// TIA Portal project "lab4" (V17)

(* hardware
DEVICE "S7-1200 station_1"  S7-1200 Station
   slot 0: "Rack_0"  S7-1200 Rack  Rack  V1.0
   slot 1: "PLC_1"  CPU 1214C DC/DC/DC  6ES7 214-1AG40-0XB0  V4.5
*)

// ===== PLC "PLC_1"  CPU 1214C DC/DC/DC =====

VAR_GLOBAL   // PLC tag table "Default tag table"
   "Zmienna_Int" AT %MW50 : Int;
   "Zmienna_Real" AT %MD52 : Real;
   "Zmienna_Word" AT %MW56 : Word;
   "Zmienna_UInt" AT %MW58 : UInt;
   "Zmienna_DInt" AT %MD59 : DInt;
   "Tag_1" AT %Q0.0 : Bool;
   "Tag_2" AT %M50.0 : Bool;
   "Tag_3" AT %M100.0 : Bool;
   "Tag_4" AT %M99.0 : Bool;
   "Tag_5" AT %Q0.1 : Bool;
   "Tag_6" AT %I0.0 : Bool;
   "Tag_7" AT %M0.0 : Bool;
   "Tag_8" AT %M0.1 : Bool;
   "Tag_9" AT %Q0.2 : Bool;
   "Tag_10" AT %IB0 : Byte;
   "Tag_11" AT %QB0 : Byte;
END_VAR

DATA_BLOCK "Rejestr_przesuwny_DB"   // DB6
{ S7_Optimized_Access := 'TRUE' }
VERSION : 0.1
   VAR
      Rejestr : Array[0..9] of Byte;
   END_VAR
BEGIN
END_DATA_BLOCK

// folder: System blocks/Program resources

DATA_BLOCK "IEC_Timer_0_DB"   // DB1
{ S7_Optimized_Access := 'TRUE' }
AUTHOR : Simatic
FAMILY : IEC
NAME : IEC_TMR
VERSION : 1.0
// stored: InstanceOfName IEC_TIMER
"IEC_TIMER"
BEGIN
END_DATA_BLOCK

DATA_BLOCK "IEC_Timer_0_DB_1"   // DB2
{ S7_Optimized_Access := 'TRUE' }
AUTHOR : Simatic
FAMILY : IEC
NAME : IEC_TMR
VERSION : 1.0
// stored: InstanceOfName IEC_TIMER
"IEC_TIMER"
BEGIN
END_DATA_BLOCK

DATA_BLOCK "IEC_Counter_0_DB"   // DB3
{ S7_Optimized_Access := 'TRUE' }
AUTHOR : Simatic
FAMILY : IEC
NAME : CNTR
VERSION : 1.0
// stored: InstanceOfName IEC_COUNTER
"IEC_COUNTER"
BEGIN
END_DATA_BLOCK

DATA_BLOCK "Counter_czerwone_DB"   // DB4
{ S7_Optimized_Access := 'TRUE' }
AUTHOR : Simatic
FAMILY : IEC
NAME : CNTR
VERSION : 1.0
// stored: InstanceOfName IEC_COUNTER
"IEC_COUNTER"
BEGIN
END_DATA_BLOCK

DATA_BLOCK "Counter_nieb_DB"   // DB5
{ S7_Optimized_Access := 'TRUE' }
AUTHOR : Simatic
FAMILY : IEC
NAME : CNTR
VERSION : 1.0
// stored: InstanceOfName IEC_COUNTER
"IEC_COUNTER"
BEGIN
END_DATA_BLOCK

// folder: (top level)

FUNCTION "2Hz" : Void   // FC1, LAD
{ S7_Optimized_Access := 'TRUE' }
VERSION : 0.1
   VAR_INPUT
      Okres : DInt;
      "Wypelnienie [%]" : Int;
   END_VAR
   VAR_OUTPUT
      OUT : Bool;
   END_VAR
   VAR_TEMP
      Wypelnienie_temp : DInt;
      Wypelnienie_DInt : DInt;
      TP_temp : Bool;
   END_VAR
   VAR_TEMP   // added for the SCL form of the ladder/FBD networks
      _w1 : Bool;
   END_VAR
BEGIN

REGION Network 1
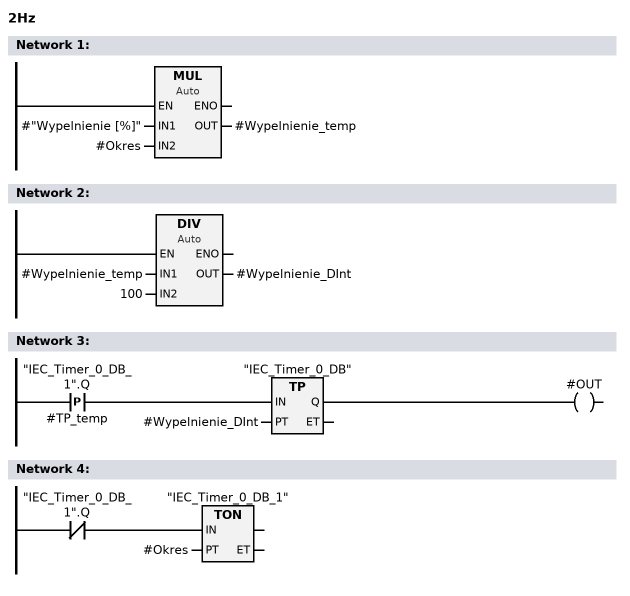
   RUNG wire#powerrail
      Mul(in1 := #"Wypelnienie [%]", in2 := #Okres, out => #Wypelnienie_temp)
   END_RUNG
   // the same network as SCL:
   #Wypelnienie_temp := #"Wypelnienie [%]" * #Okres;
END_REGION

REGION Network 2
   RUNG wire#powerrail
      Div(in1 := #Wypelnienie_temp, in2 := 100, out => #Wypelnienie_DInt)
   END_RUNG
   // the same network as SCL:
   #Wypelnienie_DInt := #Wypelnienie_temp / 100;
END_REGION

REGION Network 3
   #_w1 := "IEC_Timer_0_DB_1".Q AND NOT #TP_temp;   // rising edge of "IEC_Timer_0_DB_1".Q
   #TP_temp := "IEC_Timer_0_DB_1".Q;
   "IEC_Timer_0_DB".TP(IN := #_w1, PT := #Wypelnienie_DInt);
   #OUT := "IEC_Timer_0_DB".Q;
END_REGION

REGION Network 4
   "IEC_Timer_0_DB_1".TON(IN := NOT "IEC_Timer_0_DB_1".Q, PT := #Okres);
END_REGION
END_FUNCTION

FUNCTION "Pakowanie" : Void   // FC2, LAD
{ S7_Optimized_Access := 'TRUE' }
VERSION : 0.1
   VAR_INPUT
      Czujnik_podajnik : Bool;
      Clock : Bool;
   END_VAR
   VAR_IN_OUT
      Naped : Bool;
      Czerwony_element : Bool;
      Niebieski_element : Bool;
      Fotokomorka_nieb : Bool;
      Fotokomorka_czerw : Bool;
   END_VAR
   VAR_TEMP
      Uruchom_temp : Bool;
      Clock_temp : Bool;
      Dodaj_czerw : Bool;
      Dodaj_nieb : Bool;
   END_VAR
   VAR_TEMP   // added for the SCL form of the ladder/FBD networks
      _w1 : Bool;
   END_VAR
BEGIN

REGION Network 1
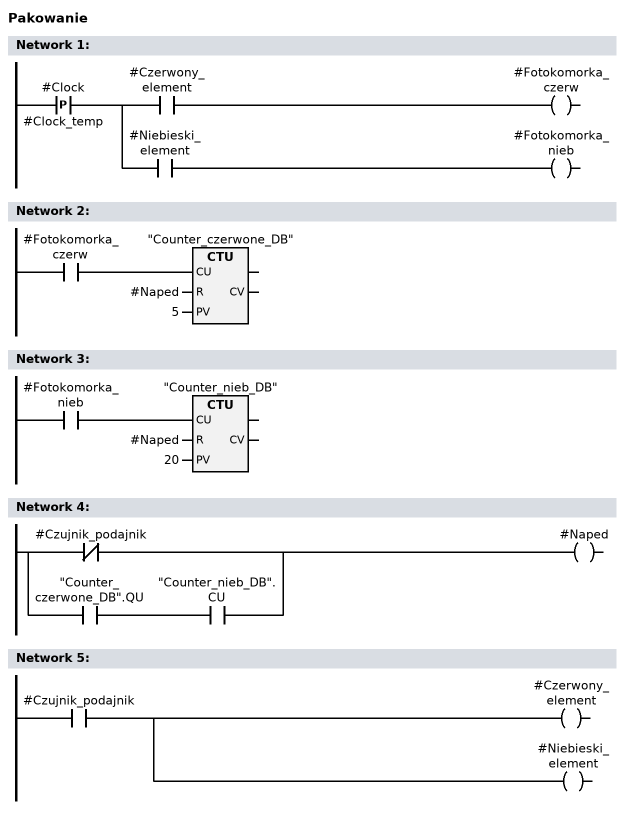
   RUNG wire#powerrail
      P_Contact(operand := #Clock, bit := #Clock_temp)
      wire#w1
      Contact( #Czerwony_element )
      Coil( #Fotokomorka_czerw )
   END_RUNG
   RUNG wire#w1
      Contact( #Niebieski_element )
      Coil( #Fotokomorka_nieb )
   END_RUNG
   // the same network as SCL:
   #_w1 := #Clock AND NOT #Clock_temp;   // rising edge of #Clock
   #Clock_temp := #Clock;
   #Fotokomorka_czerw := #_w1 AND #Czerwony_element;
   #Fotokomorka_nieb := #_w1 AND #Niebieski_element;
END_REGION

REGION Network 2
   "Counter_czerwone_DB".CTU(CU := #Fotokomorka_czerw, R := #Naped, PV := 5);
END_REGION

REGION Network 3
   "Counter_nieb_DB".CTU(CU := #Fotokomorka_nieb, R := #Naped, PV := 20);
END_REGION

REGION Network 4
   RUNG wire#powerrail
      I_Contact( #Czujnik_podajnik )
      wire#w1
      Coil( #Naped )
   END_RUNG
   RUNG wire#powerrail
      Contact( "Counter_czerwone_DB".QU )
      Contact( "Counter_nieb_DB".CU )
   END_RUNG wire#w1
   // the same network as SCL:
   #Naped := NOT #Czujnik_podajnik OR ("Counter_czerwone_DB".QU AND "Counter_nieb_DB".CU);
END_REGION

REGION Network 5
   RUNG wire#powerrail
      Contact( #Czujnik_podajnik )
      wire#w1
      Coil( #Czerwony_element )
   END_RUNG
   RUNG wire#w1
      Coil( #Niebieski_element )
   END_RUNG
   // the same network as SCL:
   #Czerwony_element := #Czujnik_podajnik;
   #Niebieski_element := #Czujnik_podajnik;
END_REGION
END_FUNCTION

FUNCTION "Dzielnik_4_1" : Void   // FC3, LAD
{ S7_Optimized_Access := 'TRUE' }
VERSION : 0.1
   VAR_INPUT
      Signal_IN : Bool;
   END_VAR
   VAR_OUTPUT
      Signal_Out : Bool;
   END_VAR
BEGIN

REGION Network 1
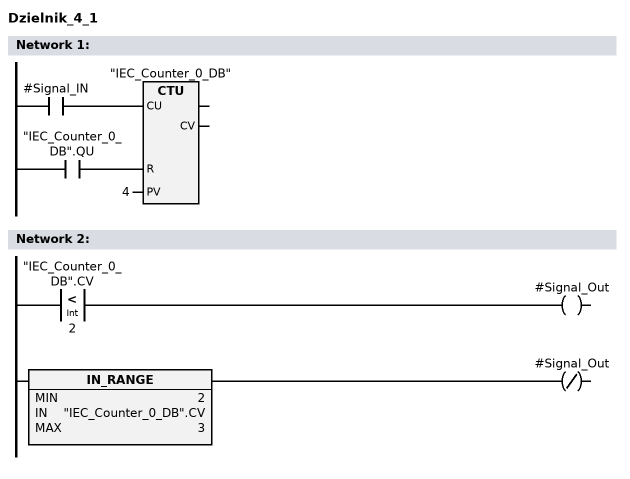
   "IEC_Counter_0_DB".CTU(CU := #Signal_IN, R := "IEC_Counter_0_DB".QU, PV := 4);
END_REGION

REGION Network 2
   RUNG wire#powerrail
      { S7_Templates := "SrcType := Int" } LT_Contact(in1 := "IEC_Counter_0_DB".CV, in2 := 2)
      Coil( #Signal_Out )
   END_RUNG
   RUNG wire#powerrail
      { S7_Templates := "SrcType := Int" } InRange(min := 2, in := "IEC_Counter_0_DB".CV, max := 3)
      I_Coil( #Signal_Out )
   END_RUNG
   // the same network as SCL:
   #Signal_Out := "IEC_Counter_0_DB".CV < 2;
   #Signal_Out := NOT ((2 <= "IEC_Counter_0_DB".CV) AND ("IEC_Counter_0_DB".CV <= 3));
END_REGION
END_FUNCTION

FUNCTION "Rejestr_przesuwny" : Void   // FC4, LAD
{ S7_Optimized_Access := 'TRUE' }
VERSION : 0.1
   VAR_INPUT
      Clock : Bool;
   END_VAR
   VAR_TEMP
      Clock_temp : Bool;
   END_VAR
   VAR_TEMP   // added for the SCL form of the ladder/FBD networks
      _w1 : Bool;
   END_VAR
BEGIN

REGION Network 1
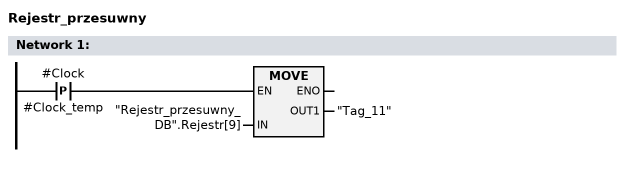
   RUNG wire#powerrail
      P_Contact(operand := #Clock, bit := #Clock_temp)
      Move(in := "Rejestr_przesuwny_DB".Rejestr[9], out1 => "Tag_11")
   END_RUNG
   // the same network as SCL:
   #_w1 := #Clock AND NOT #Clock_temp;   // rising edge of #Clock
   #Clock_temp := #Clock;
   IF #_w1 THEN "Tag_11" := "Rejestr_przesuwny_DB".Rejestr[9]; END_IF;
END_REGION
END_FUNCTION

ORGANIZATION_BLOCK "Main"   // OB1, LAD, ProgramCycle
TITLE = "Main Program Sweep (Cycle)"
{ S7_Optimized_Access := 'TRUE' }
VERSION : 0.1
   VAR_INPUT
      Initial_Call : Bool;   // Initial call of this OB
      Remanence : Bool;   // =True, if remanent data are available
   END_VAR
BEGIN

REGION Network 1
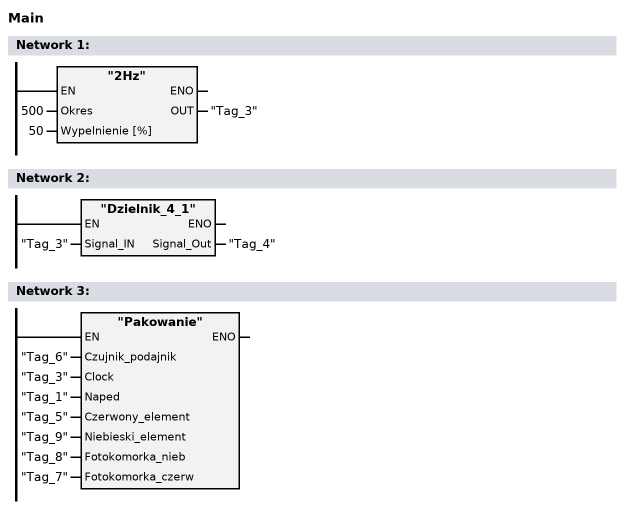
   RUNG wire#powerrail
      "2Hz"(Okres := 500, "Wypelnienie [%]" := 50, OUT => "Tag_3")
   END_RUNG
   // the same network as SCL:
   "2Hz"(Okres := 500, "Wypelnienie [%]" := 50, OUT => "Tag_3");
END_REGION

REGION Network 2
   RUNG wire#powerrail
      "Dzielnik_4_1"(Signal_IN := "Tag_3", Signal_Out => "Tag_4")
   END_RUNG
   // the same network as SCL:
   "Dzielnik_4_1"(Signal_IN := "Tag_3", Signal_Out => "Tag_4");
END_REGION

REGION Network 3
   RUNG wire#powerrail
      "Pakowanie"(Czujnik_podajnik := "Tag_6", Clock := "Tag_3", Naped := "Tag_1", Czerwony_element := "Tag_5", Niebieski_element := "Tag_9", Fotokomorka_nieb := "Tag_8", Fotokomorka_czerw := "Tag_7")
   END_RUNG
   // the same network as SCL:
   "Pakowanie"(Czujnik_podajnik := "Tag_6",
               Clock := "Tag_3",
               Naped := "Tag_1",
               Czerwony_element := "Tag_5",
               Niebieski_element := "Tag_9",
               Fotokomorka_nieb := "Tag_8",
               Fotokomorka_czerw := "Tag_7");
END_REGION
END_ORGANIZATION_BLOCK

ORGANIZATION_BLOCK "Startup"   // OB100, LAD, Startup
TITLE = "Complete Restart"
{ S7_Optimized_Access := 'TRUE' }
VERSION : 0.1
   VAR_INPUT
      LostRetentive : Bool;   // True if retentive data are lost
      LostRTC : Bool;   // True if date and time are lost
   END_VAR
BEGIN

REGION Network 1
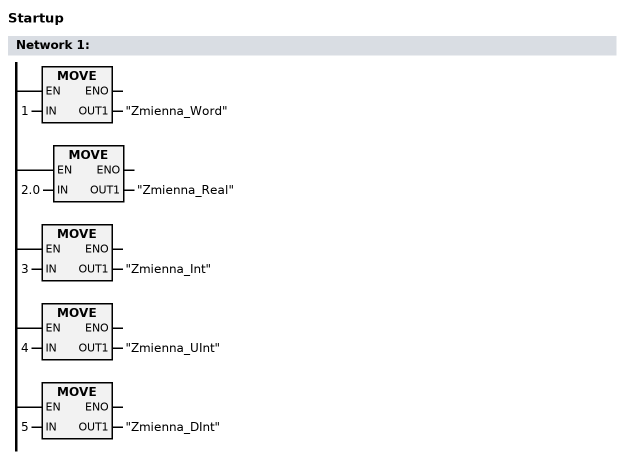
   RUNG wire#powerrail
      Move(in := 1, out1 => "Zmienna_Word")
   END_RUNG
   RUNG wire#powerrail
      Move(in := 2.0, out1 => "Zmienna_Real")
   END_RUNG
   RUNG wire#powerrail
      Move(in := 3, out1 => "Zmienna_Int")
   END_RUNG
   RUNG wire#powerrail
      Move(in := 4, out1 => "Zmienna_UInt")
   END_RUNG
   RUNG wire#powerrail
      Move(in := 5, out1 => "Zmienna_DInt")
   END_RUNG
   // the same network as SCL:
   "Zmienna_Word" := 1;
   "Zmienna_Real" := 2.0;
   "Zmienna_Int" := 3;
   "Zmienna_UInt" := 4;
   "Zmienna_DInt" := 5;
END_REGION
END_ORGANIZATION_BLOCK